{attribute 'qualified_only'}
{attribute 'strict'}
{attribute 'to_string'}
TYPE EventsEnum :
(
	//standard operation
	BUNDLE_ADDED_TO_PRODUCTION,
	BUNDLE_RECEIVED,
	BUNDLE_COMPLETE,
	
	//area complete
	AREA_1_COMPLETE,
	AREA_2_COMPLETE,
	AREA_3_COMPLETE,
	AREA_4_COMPLETE,
	AREA_5_COMPLETE,
	AREA_6_COMPLETE,
	
	//area complete
	AREA_1_RECEIVE,
	AREA_2_RECEIVE,
	AREA_3_RECEIVE,
	AREA_4_RECEIVE,
	AREA_5_RECEIVE,
	AREA_6_RECEIVE,

	//standard errors
	BACKLOG,
	MACHINE_FAILURE,
	BUNDLE_EARLY_RECEIVED,
	BUNDLE_LATE_RECEIVED,
	
	AREA_1_DELAY,
	AREA_2_DELAY,
	AREA_3_DELAY,
	AREA_4_DELAY,
	AREA_5_DELAY,
	AREA_6_DELAY,
	
	//robots, motors, database, connections, etc
	CONNECTION_ERROR_PRODUCTION_LOG,
	CONNECTION_ERROR_RECIPE_DB,
	
	CONNECTION_ERROR_AREA_1_DB,
	CONNECTION_ERROR_AREA_2_DB,
	CONNECTION_ERROR_AREA_3_DB,
	CONNECTION_ERROR_AREA_4_DB,
	CONNECTION_ERROR_AREA_5_DB,
	CONNECTION_ERROR_AREA_6_DB,
	
	size
);
END_TYPE

(* stored: Version 1.1.0.1, ProductVersion 3.1.4024.11
   EnumerationTextList EventsEnum: Id {7116f09d-954e-4b54-827f-4a9cf285982d} *)
